(* IEC 61131-3 sources: eCockpitGit/test_project/src/%PLC%PLCTest2/%PLOG%Plc Logic/%APP%APP1_Test, 6 files *)

(* ---- %DUT%enum_test.st ---- *)
{attribute 'qualified_only'}
{attribute 'strict'}
TYPE enum_test :
(
	enum1,
	enum2,
	enum3 := 5
);
END_TYPE

(* ---- %DUT%struct_test.st ---- *)
TYPE struct_test :
STRUCT
	structMember1		:BOOL;
	structMember2		:INT;
	structMember3		:STRING;
	structMember4		:WORD;
END_STRUCT
END_TYPE

(* ---- %GVL%Modbus.st ---- *)
{attribute 'qualified_only'}
VAR_GLOBAL
END_VAR

(* ---- %PV%PERSIVARS.st ---- *)
{attribute 'qualified_only'}
VAR_GLOBAL PERSISTENT RETAIN
	test1: BOOL;
	test2: INT;
END_VAR

(* ---- %POU%func_test.st ---- *)
FUNCTION func_test : BOOL
VAR_INPUT
END_VAR
VAR
END_VAR

(*%!%__DELIMITER__%!%*)

(* ---- %POU%fb_test.st ---- *)
FUNCTION_BLOCK fb_test
VAR_INPUT
END_VAR
VAR_OUTPUT
END_VAR
VAR
END_VAR

(*%!%__DELIMITER__%!%*)
